RoboDK station: Assistive_UR5e.rdk

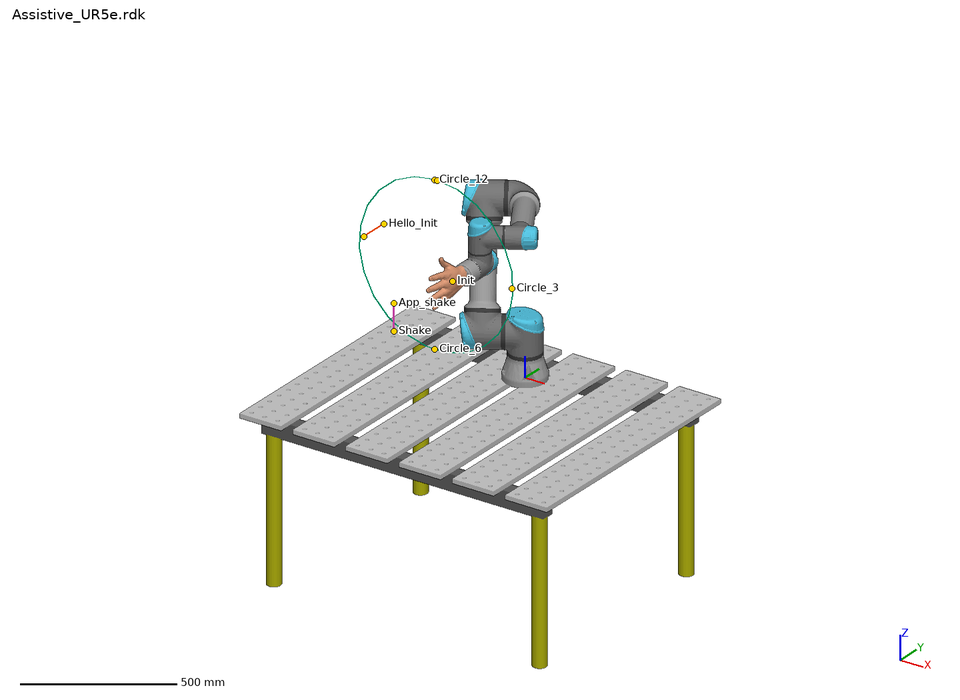
[picture v0: the station drawn from its stored meshes, robots at their saved joint values, targets as dots, program paths as lines]
Station Assistive_UR5e_SW (saved by RoboDK 5.9.2). Poses are relative to the parent item; angles as X-Y-Z fixed-axis rotations.
  - frame UR5e Base at (0, 0, 0) mm
    - robot UR5e: 6 axes, payload 5 kg, reach 850 mm, repeatability 0.03 mm, weight 18.4 kg
        modified DH rows (alpha deg, a mm, theta deg, d mm): 0, 0, 0, 162.5; 90, 0, 180, 0; 0, 425, 0, 0; 0, 392.25, 0, 133.3; -90, 0, 0, 99.7; 90, 0, 180, 99.6
        joint limits [-360, -360, -360, -360, -360, -360] to [360, 360, 360, 360, 360, 360]; home [0, -90, -90, 0, 90, 0]; saved at [-57.836, -65.392, -107.167, 172.559, -57.836, 0]
      - tool Hand, TCP at (0, 0, 50) mm, size 54.8 x 155.9 x 193.5 mm, geometry from Hand.stl
  - frame World at (0, 0, 0) mm
    - object Table at (0, 0, 0) mm, size 1193.8 x 965.2 x 609.6 mm, geometry from welding_table.sld
    - target Init (Cartesian target) at (0, -400, 500) mm, rotated rx 90 ry 0 rz 0 deg; joints [-57.836, -65.392, -107.167, 172.559, -57.836, 0] of UR5e
    - target App_shake (joint target) at (-300, -300, 300) mm, rotated rx 90 ry 0 rz 0 deg; joints [-129.97, -84.968, -123.366, -151.667, -129.97, 0] of UR5e
    - target Shake (joint target) at (-300, -300, 200) mm, rotated rx 90 ry 0 rz 0 deg; joints [-129.97, -95.332, -131.473, -133.195, -129.97, 0] of UR5e
    - target Hello_Init (joint target) at (-380.86, -238.62, 533.82) mm, rotated rx 0 ry 0 rz 90 deg; joints [-130.679, -89.195, -122.013, 301.208, -90, 130.679] of UR5e
    - target Hello_L (Cartesian target) at (-380.86, -238.62, 533.82) mm, rotated rx -27.5 ry 0 rz 90 deg; joints [-122.724, -77.892, -124.578, 276.752, -67.141, 125.921] of UR5e
    - target Hello_R (Cartesian target) at (-380.86, -238.62, 533.82) mm, rotated rx 35 ry 0 rz 90 deg; joints [-138.185, -102.099, -110.776, 330.433, -112.484, 143.766] of UR5e
    - target Give5 (Cartesian target) at (-380.86, -350, 533.82) mm, rotated rx 0 ry 0 rz 90 deg; joints [-122.484, -98.377, -112.067, 300.444, -90, 122.484] of UR5e
    - target Circle_12 (Cartesian target) at (0, -500, 900) mm, rotated rx 90 ry 0 rz 0 deg; joints [67.64, -90.732, 57.872, -147.139, -67.64, 180] of UR5e
    - target Circle_6 (Cartesian target) at (0, -500, 300) mm, rotated rx 90 ry 0 rz 0 deg; joints [67.64, -67.946, 133.155, -245.209, -67.64, 180] of UR5e
    - target Circle_3 (Cartesian target) at (300, -500, 600) mm, rotated rx 90 ry 0 rz 0 deg; joints [113.772, -82.119, 94.363, -192.244, -113.772, 180] of UR5e
    - target Circle~12 (Cartesian target) at (10, -500, 900) mm, rotated rx 90 ry 0 rz 0 deg; joints [69.284, -90.712, 57.851, -147.14, -69.284, 180] of UR5e
  - program Init (3 instructions, listed below)
  - program Hello (8 instructions, listed below)
  - program Give_me_5! (5 instructions, listed below)
  - program Circle (4 instructions, listed below)
  - program Hand_shake (5 instructions, listed below)
  - program MainProgram (6 instructions, listed below)
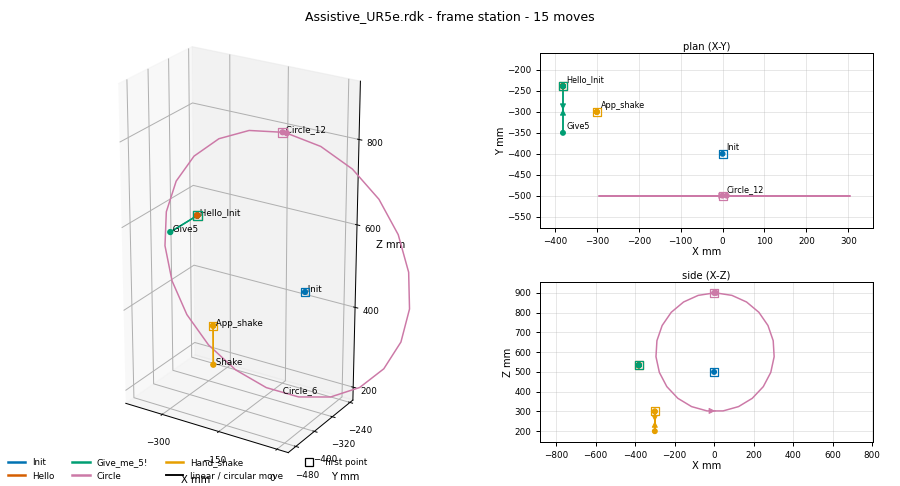
[picture p0: tool path of Assistive_UR5e.rdk in frame station, 15 of 15 moves have a stored position in this frame; points joined in program order, loops and branches not executed]

--- program Init (robot UR5e) ---
  Est. Ref.: UR5e Base
  Est. herr: Hand
  MoveJ (Init)

--- program Hello (robot UR5e) ---
  Set Ref.: World
  Set Tool: Hand
  MoveJ (Hello_Init)
  MoveL (Hello_L)
  MoveL (Hello_R)
  MoveL (Hello_L)
  MoveL (Hello_R)
  MoveL (Hello_Init)

--- program Give_me_5! (robot UR5e) ---
  Est. Ref.: UR5e Base
  Est. herr: Hand
  MoveL (App_give5) -> target Hello_Init
  MoveL (Give5)
  MoveL (App_give5) -> target Hello_Init

--- program Circle (robot UR5e) ---
  Set Ref.: World
  Set Tool: Hand
  MoveJ (Circle_12)
  MoveC (Circle_6, Circle~12)

--- program Hand_shake (robot UR5e) ---
  Est. Ref.: UR5e Base
  Est. herr: Hand
  MoveL (App_shake)
  MoveL (Shake)
  MoveL (App_shake)

--- program MainProgram (robot UR5e) ---
  Llamar Init
  Call Hello
  Llamar Hand_shake
  Llamar Give_me_5!
  Call Circle
  Llamar Init
